PROGRAM Agitadores
VAR
	PP1_L1_AG: Equipo_Motor_No_Rev;
	wPP1_L1_AG_HoraIni:INT;
	wPP1_L1_AG_CantHora:INT;
	wPP1_L1_AG_HoraFin:INT;
	bPP1_L1_AG_ResetAl: BOOL;	
	//
	PP1_L2_AG: Equipo_Motor_No_Rev;
	wPP1_L2_AG_HoraIni:INT;
	wPP1_L2_AG_CantHora:INT;
	wPP1_L2_AG_HoraFin:INT;
	//
	PP1_L3_AG: Equipo_Motor_No_Rev;
	wPP1_L3_AG_HoraIni:INT;
	wPP1_L3_AG_CantHora:INT;
	wPP1_L3_AG_HoraFin:INT;	
	//
	PP1_L4_AG: Equipo_Motor_No_Rev;
	wPP1_L4_AG_HoraIni:INT;
	wPP1_L4_AG_CantHora:INT;
	wPP1_L4_AG_HoraFin:INT;	
	//	
	PP2_L5_AG: Equipo_Motor_No_Rev;
	wPP2_L5_AG_HoraIni:INT;
	wPP2_L5_AG_CantHora:INT;
	wPP2_L5_AG_HoraFin:INT;
	bPP2_L5_AG_ResetAl: BOOL;	
	//
	PP2_L6_AG: Equipo_Motor_No_Rev;
	wPP2_L6_AG_HoraIni:INT;
	wPP2_L6_AG_CantHora:INT;
	wPP2_L6_AG_HoraFin:INT;	
	//
	PP2_L7_AG: Equipo_Motor_No_Rev;
	wPP2_L7_AG_HoraIni:INT;
	wPP2_L7_AG_CantHora:INT;
	wPP2_L7_AG_HoraFin:INT;	
	//
	PP2_L8_AG: Equipo_Motor_No_Rev;
	wPP2_L8_AG_HoraIni:INT;
	wPP2_L8_AG_CantHora:INT;
	wPP2_L8_AG_HoraFin:INT;
	//
	PP3_L9_AG: Equipo_Motor_No_Rev;
	wPP3_L9_AG_HoraIni:INT;
	wPP3_L9_AG_CantHora:INT;
	wPP3_L9_AG_HoraFin:INT;	
	//
	PP3_L10_AG: Equipo_Motor_No_Rev;
	wPP3_L10_AG_HoraIni:INT;
	wPP3_L10_AG_CantHora:INT;
	wPP3_L10_AG_HoraFin:INT;	
	//
	PP3_L11_AG: Equipo_Motor_No_Rev;
	wPP3_L11_AG_HoraIni:INT;
	wPP3_L11_AG_CantHora:INT;
	wPP3_L11_AG_HoraFin:INT;	
	//
	PP3_L12_AG: Equipo_Motor_No_Rev;
	wPP3_L12_AG_HoraIni:INT;
	wPP3_L12_AG_CantHora:INT;
	wPP3_L12_AG_HoraFin:INT;	
END_VAR

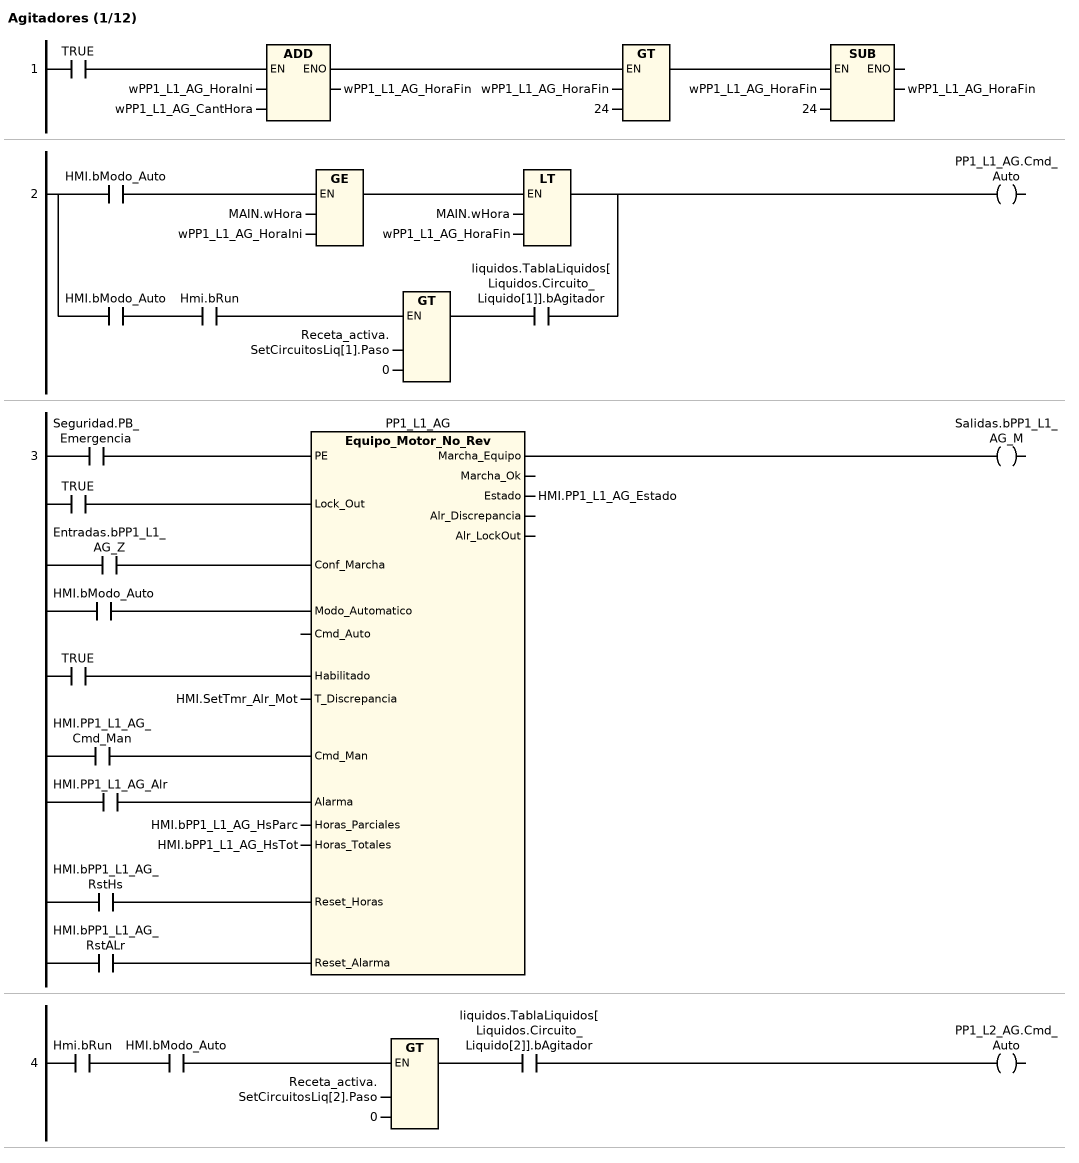
// NETWORK 1
wPP1_L1_AG_HoraFin := wPP1_L1_AG_HoraIni + wPP1_L1_AG_CantHora;
IF wPP1_L1_AG_HoraFin > 24 THEN wPP1_L1_AG_HoraFin := wPP1_L1_AG_HoraFin - 24; END_IF

// NETWORK 2
PP1_L1_AG.Cmd_Auto := HMI.bModo_Auto AND MAIN.wHora >= wPP1_L1_AG_HoraIni AND MAIN.wHora < wPP1_L1_AG_HoraFin OR (HMI.bModo_Auto AND Hmi.bRun AND Receta_activa.SetCircuitosLiq[1].Paso > 0) AND (liquidos.TablaLiquidos[Liquidos.Circuito_Liquido[1]].bAgitador);

// NETWORK 3
PP1_L1_AG(
    PE := Seguridad.PB_Emergencia,
    Lock_Out := TRUE,
    Conf_Marcha := Entradas.bPP1_L1_AG_Z,
    Modo_Automatico := HMI.bModo_Auto,
    Habilitado := TRUE,
    T_Discrepancia := HMI.SetTmr_Alr_Mot,
    Cmd_Man := HMI.PP1_L1_AG_Cmd_Man,
    Alarma := HMI.PP1_L1_AG_Alr,
    Horas_Parciales := HMI.bPP1_L1_AG_HsParc,
    Horas_Totales := HMI.bPP1_L1_AG_HsTot,
    Reset_Horas := HMI.bPP1_L1_AG_RstHs,
    Reset_Alarma := HMI.bPP1_L1_AG_RstALr,
    Estado => HMI.PP1_L1_AG_Estado); // Equipo_Motor_No_Rev
Salidas.bPP1_L1_AG_M := PP1_L1_AG.Marcha_Equipo;

// NETWORK 4
PP1_L2_AG.Cmd_Auto := (Hmi.bRun AND HMI.bModo_Auto AND Receta_activa.SetCircuitosLiq[2].Paso > 0) AND (liquidos.TablaLiquidos[Liquidos.Circuito_Liquido[2]].bAgitador);

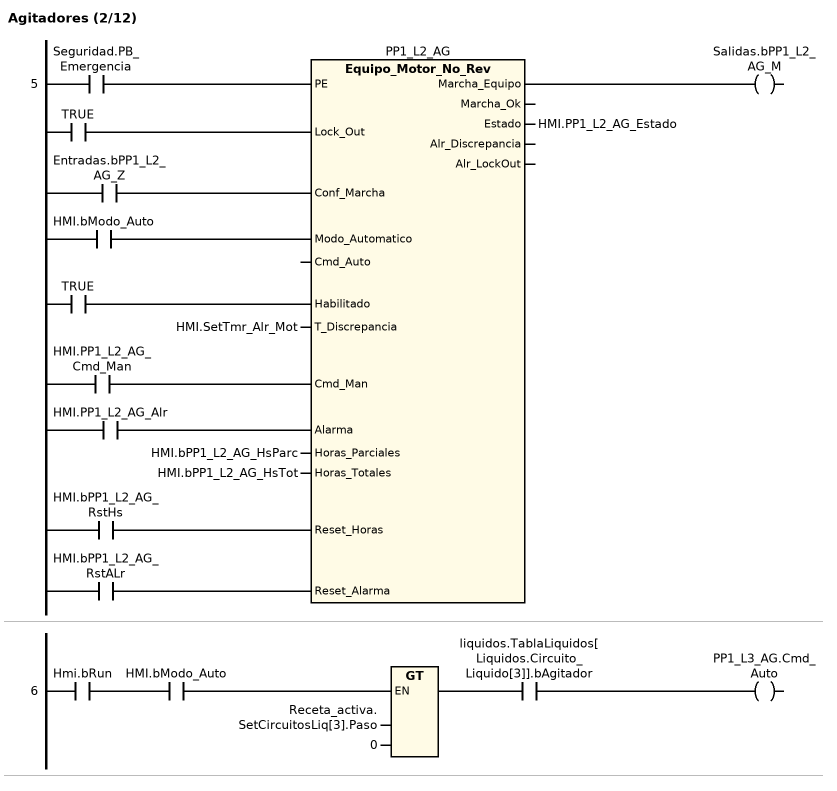
// NETWORK 5
PP1_L2_AG(
    PE := Seguridad.PB_Emergencia,
    Lock_Out := TRUE,
    Conf_Marcha := Entradas.bPP1_L2_AG_Z,
    Modo_Automatico := HMI.bModo_Auto,
    Habilitado := TRUE,
    T_Discrepancia := HMI.SetTmr_Alr_Mot,
    Cmd_Man := HMI.PP1_L2_AG_Cmd_Man,
    Alarma := HMI.PP1_L2_AG_Alr,
    Horas_Parciales := HMI.bPP1_L2_AG_HsParc,
    Horas_Totales := HMI.bPP1_L2_AG_HsTot,
    Reset_Horas := HMI.bPP1_L2_AG_RstHs,
    Reset_Alarma := HMI.bPP1_L2_AG_RstALr,
    Estado => HMI.PP1_L2_AG_Estado); // Equipo_Motor_No_Rev
Salidas.bPP1_L2_AG_M := PP1_L2_AG.Marcha_Equipo;

// NETWORK 6
PP1_L3_AG.Cmd_Auto := (Hmi.bRun AND HMI.bModo_Auto AND Receta_activa.SetCircuitosLiq[3].Paso > 0) AND (liquidos.TablaLiquidos[Liquidos.Circuito_Liquido[3]].bAgitador);

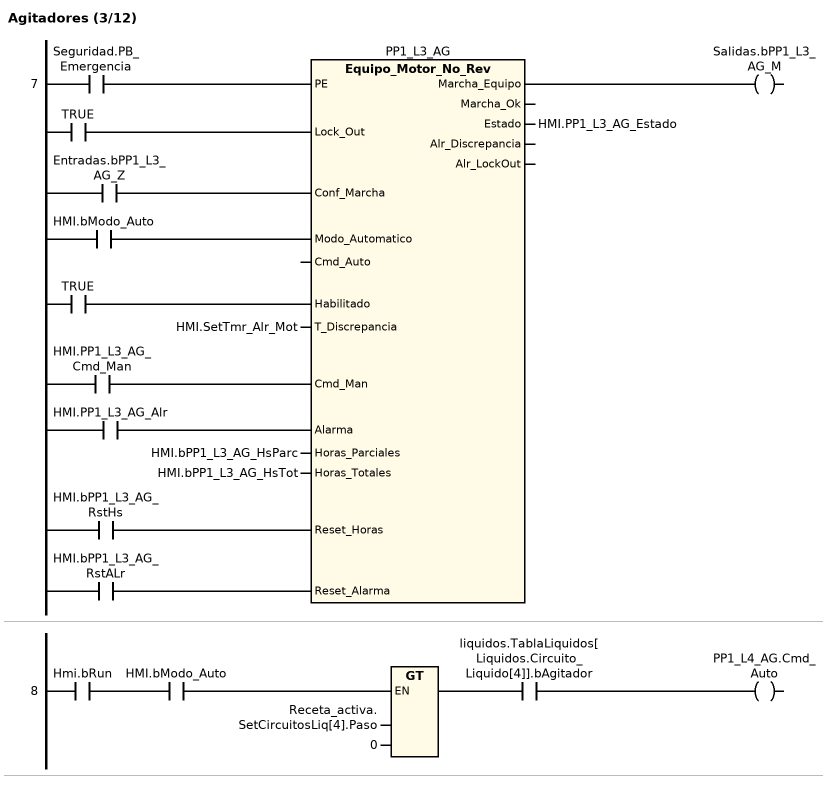
// NETWORK 7
PP1_L3_AG(
    PE := Seguridad.PB_Emergencia,
    Lock_Out := TRUE,
    Conf_Marcha := Entradas.bPP1_L3_AG_Z,
    Modo_Automatico := HMI.bModo_Auto,
    Habilitado := TRUE,
    T_Discrepancia := HMI.SetTmr_Alr_Mot,
    Cmd_Man := HMI.PP1_L3_AG_Cmd_Man,
    Alarma := HMI.PP1_L3_AG_Alr,
    Horas_Parciales := HMI.bPP1_L3_AG_HsParc,
    Horas_Totales := HMI.bPP1_L3_AG_HsTot,
    Reset_Horas := HMI.bPP1_L3_AG_RstHs,
    Reset_Alarma := HMI.bPP1_L3_AG_RstALr,
    Estado => HMI.PP1_L3_AG_Estado); // Equipo_Motor_No_Rev
Salidas.bPP1_L3_AG_M := PP1_L3_AG.Marcha_Equipo;

// NETWORK 8
PP1_L4_AG.Cmd_Auto := (Hmi.bRun AND HMI.bModo_Auto AND Receta_activa.SetCircuitosLiq[4].Paso > 0) AND (liquidos.TablaLiquidos[Liquidos.Circuito_Liquido[4]].bAgitador);

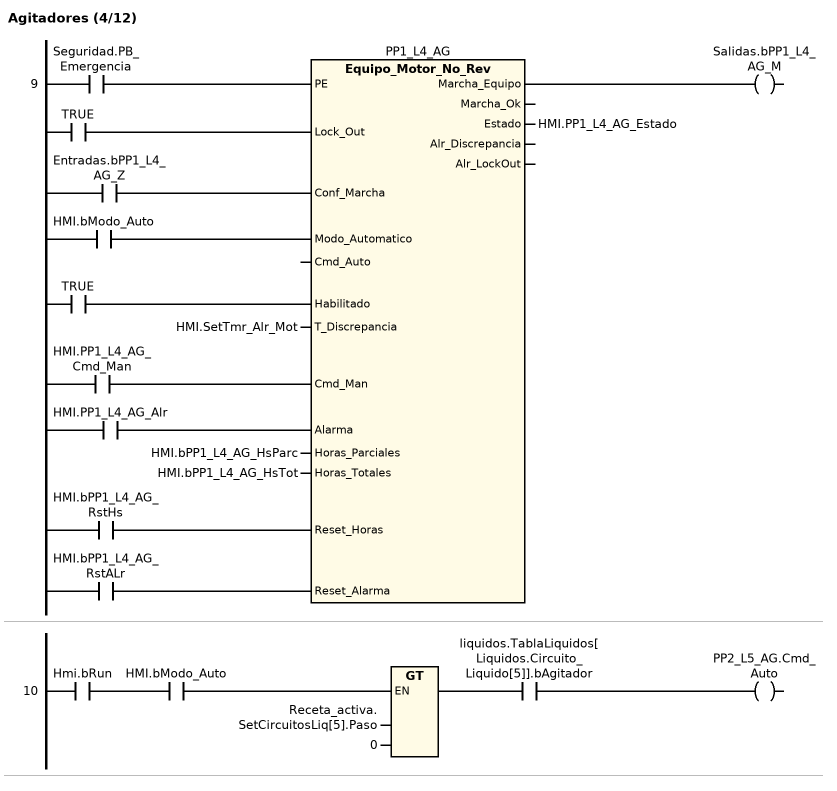
// NETWORK 9
PP1_L4_AG(
    PE := Seguridad.PB_Emergencia,
    Lock_Out := TRUE,
    Conf_Marcha := Entradas.bPP1_L4_AG_Z,
    Modo_Automatico := HMI.bModo_Auto,
    Habilitado := TRUE,
    T_Discrepancia := HMI.SetTmr_Alr_Mot,
    Cmd_Man := HMI.PP1_L4_AG_Cmd_Man,
    Alarma := HMI.PP1_L4_AG_Alr,
    Horas_Parciales := HMI.bPP1_L4_AG_HsParc,
    Horas_Totales := HMI.bPP1_L4_AG_HsTot,
    Reset_Horas := HMI.bPP1_L4_AG_RstHs,
    Reset_Alarma := HMI.bPP1_L4_AG_RstALr,
    Estado => HMI.PP1_L4_AG_Estado); // Equipo_Motor_No_Rev
Salidas.bPP1_L4_AG_M := PP1_L4_AG.Marcha_Equipo;

// NETWORK 10
PP2_L5_AG.Cmd_Auto := (Hmi.bRun AND HMI.bModo_Auto AND Receta_activa.SetCircuitosLiq[5].Paso > 0) AND (liquidos.TablaLiquidos[Liquidos.Circuito_Liquido[5]].bAgitador);

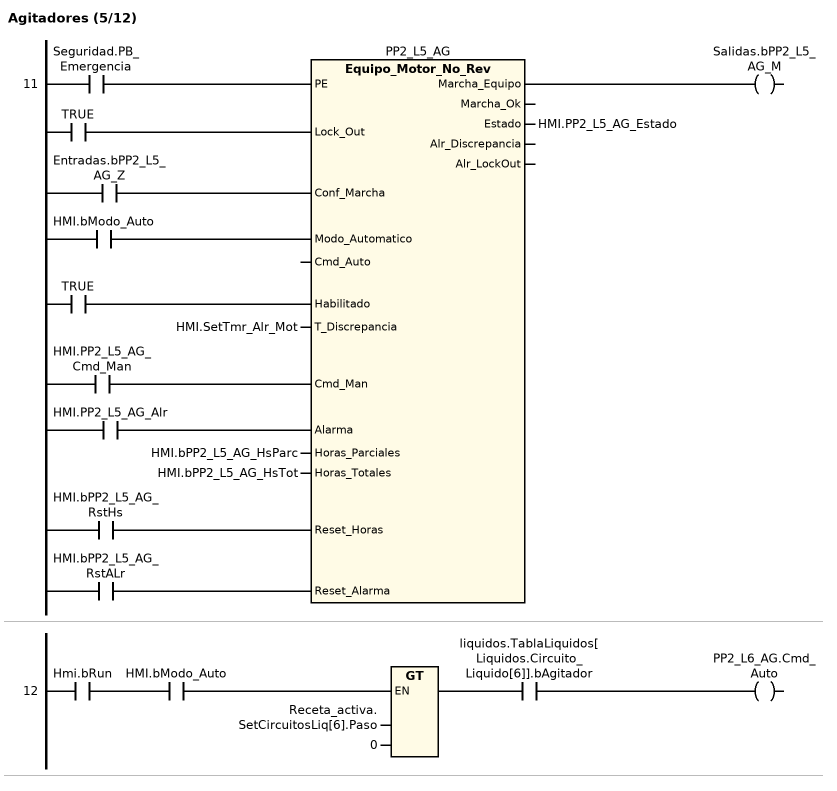
// NETWORK 11
PP2_L5_AG(
    PE := Seguridad.PB_Emergencia,
    Lock_Out := TRUE,
    Conf_Marcha := Entradas.bPP2_L5_AG_Z,
    Modo_Automatico := HMI.bModo_Auto,
    Habilitado := TRUE,
    T_Discrepancia := HMI.SetTmr_Alr_Mot,
    Cmd_Man := HMI.PP2_L5_AG_Cmd_Man,
    Alarma := HMI.PP2_L5_AG_Alr,
    Horas_Parciales := HMI.bPP2_L5_AG_HsParc,
    Horas_Totales := HMI.bPP2_L5_AG_HsTot,
    Reset_Horas := HMI.bPP2_L5_AG_RstHs,
    Reset_Alarma := HMI.bPP2_L5_AG_RstALr,
    Estado => HMI.PP2_L5_AG_Estado); // Equipo_Motor_No_Rev
Salidas.bPP2_L5_AG_M := PP2_L5_AG.Marcha_Equipo;

// NETWORK 12
PP2_L6_AG.Cmd_Auto := (Hmi.bRun AND HMI.bModo_Auto AND Receta_activa.SetCircuitosLiq[6].Paso > 0) AND (liquidos.TablaLiquidos[Liquidos.Circuito_Liquido[6]].bAgitador);

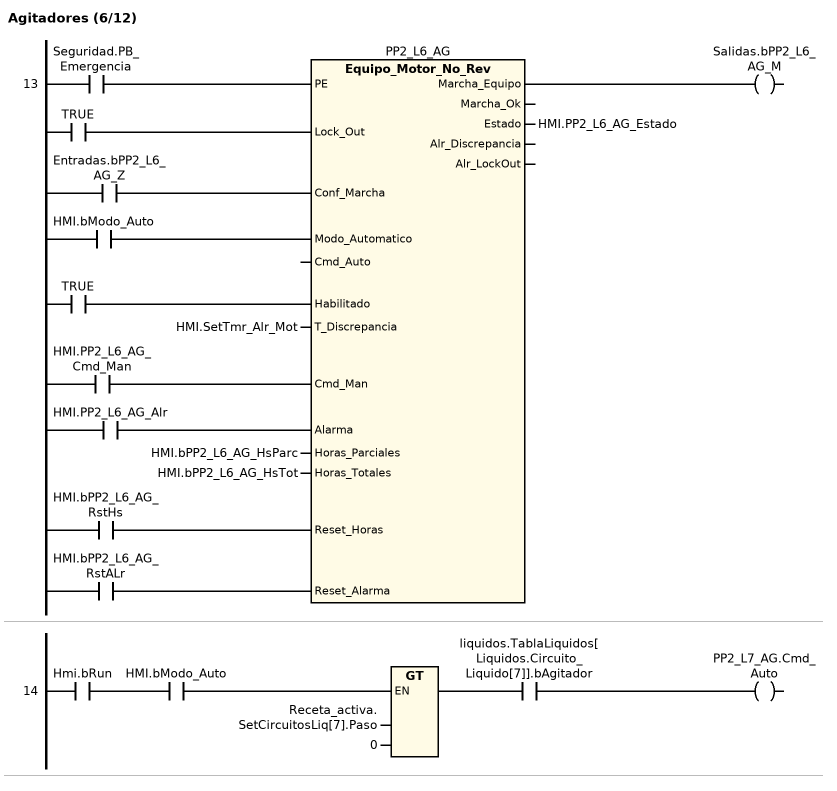
// NETWORK 13
PP2_L6_AG(
    PE := Seguridad.PB_Emergencia,
    Lock_Out := TRUE,
    Conf_Marcha := Entradas.bPP2_L6_AG_Z,
    Modo_Automatico := HMI.bModo_Auto,
    Habilitado := TRUE,
    T_Discrepancia := HMI.SetTmr_Alr_Mot,
    Cmd_Man := HMI.PP2_L6_AG_Cmd_Man,
    Alarma := HMI.PP2_L6_AG_Alr,
    Horas_Parciales := HMI.bPP2_L6_AG_HsParc,
    Horas_Totales := HMI.bPP2_L6_AG_HsTot,
    Reset_Horas := HMI.bPP2_L6_AG_RstHs,
    Reset_Alarma := HMI.bPP2_L6_AG_RstALr,
    Estado => HMI.PP2_L6_AG_Estado); // Equipo_Motor_No_Rev
Salidas.bPP2_L6_AG_M := PP2_L6_AG.Marcha_Equipo;

// NETWORK 14
PP2_L7_AG.Cmd_Auto := (Hmi.bRun AND HMI.bModo_Auto AND Receta_activa.SetCircuitosLiq[7].Paso > 0) AND (liquidos.TablaLiquidos[Liquidos.Circuito_Liquido[7]].bAgitador);

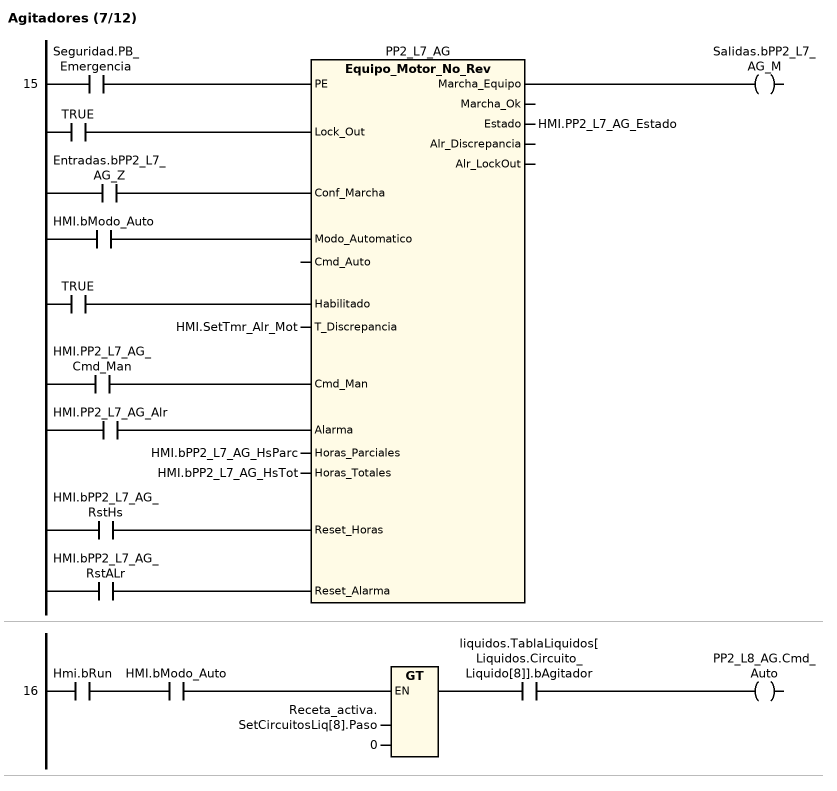
// NETWORK 15
PP2_L7_AG(
    PE := Seguridad.PB_Emergencia,
    Lock_Out := TRUE,
    Conf_Marcha := Entradas.bPP2_L7_AG_Z,
    Modo_Automatico := HMI.bModo_Auto,
    Habilitado := TRUE,
    T_Discrepancia := HMI.SetTmr_Alr_Mot,
    Cmd_Man := HMI.PP2_L7_AG_Cmd_Man,
    Alarma := HMI.PP2_L7_AG_Alr,
    Horas_Parciales := HMI.bPP2_L7_AG_HsParc,
    Horas_Totales := HMI.bPP2_L7_AG_HsTot,
    Reset_Horas := HMI.bPP2_L7_AG_RstHs,
    Reset_Alarma := HMI.bPP2_L7_AG_RstALr,
    Estado => HMI.PP2_L7_AG_Estado); // Equipo_Motor_No_Rev
Salidas.bPP2_L7_AG_M := PP2_L7_AG.Marcha_Equipo;

// NETWORK 16
PP2_L8_AG.Cmd_Auto := (Hmi.bRun AND HMI.bModo_Auto AND Receta_activa.SetCircuitosLiq[8].Paso > 0) AND (liquidos.TablaLiquidos[Liquidos.Circuito_Liquido[8]].bAgitador);

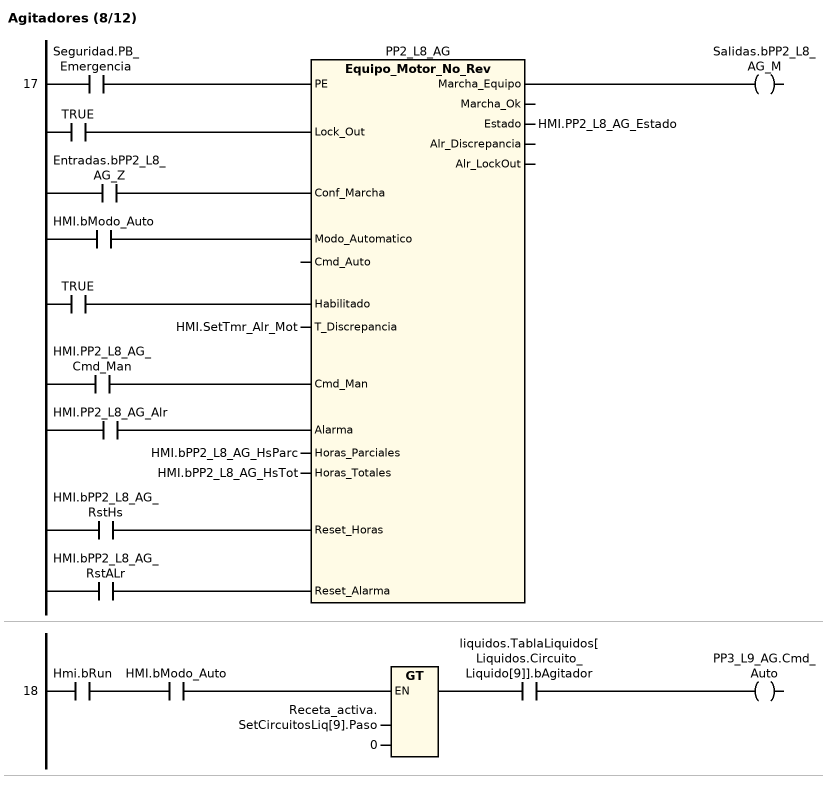
// NETWORK 17
PP2_L8_AG(
    PE := Seguridad.PB_Emergencia,
    Lock_Out := TRUE,
    Conf_Marcha := Entradas.bPP2_L8_AG_Z,
    Modo_Automatico := HMI.bModo_Auto,
    Habilitado := TRUE,
    T_Discrepancia := HMI.SetTmr_Alr_Mot,
    Cmd_Man := HMI.PP2_L8_AG_Cmd_Man,
    Alarma := HMI.PP2_L8_AG_Alr,
    Horas_Parciales := HMI.bPP2_L8_AG_HsParc,
    Horas_Totales := HMI.bPP2_L8_AG_HsTot,
    Reset_Horas := HMI.bPP2_L8_AG_RstHs,
    Reset_Alarma := HMI.bPP2_L8_AG_RstALr,
    Estado => HMI.PP2_L8_AG_Estado); // Equipo_Motor_No_Rev
Salidas.bPP2_L8_AG_M := PP2_L8_AG.Marcha_Equipo;

// NETWORK 18
PP3_L9_AG.Cmd_Auto := (Hmi.bRun AND HMI.bModo_Auto AND Receta_activa.SetCircuitosLiq[9].Paso > 0) AND (liquidos.TablaLiquidos[Liquidos.Circuito_Liquido[9]].bAgitador);

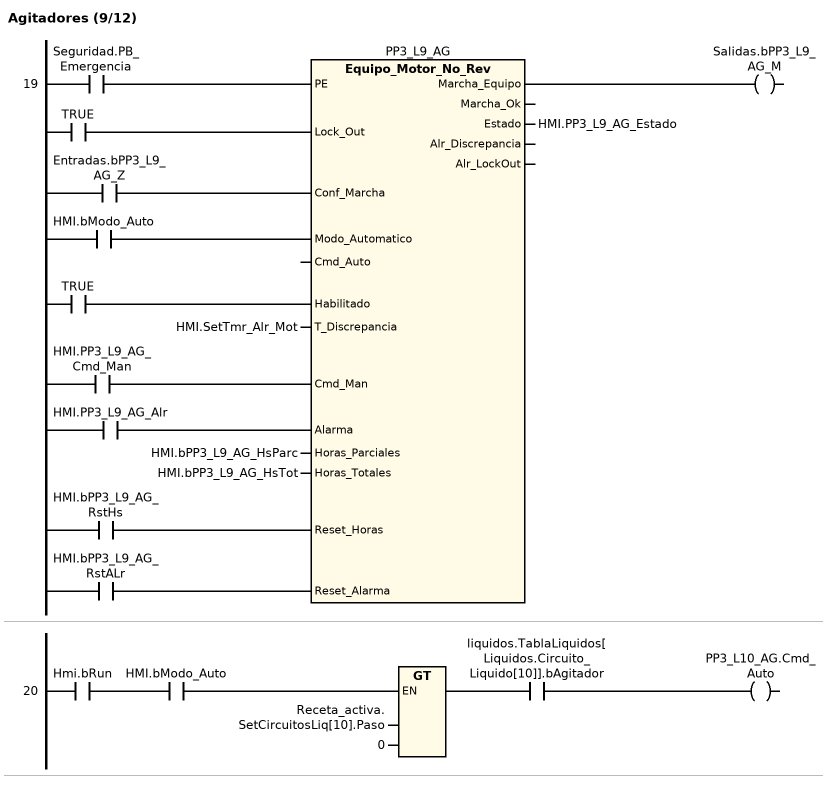
// NETWORK 19
PP3_L9_AG(
    PE := Seguridad.PB_Emergencia,
    Lock_Out := TRUE,
    Conf_Marcha := Entradas.bPP3_L9_AG_Z,
    Modo_Automatico := HMI.bModo_Auto,
    Habilitado := TRUE,
    T_Discrepancia := HMI.SetTmr_Alr_Mot,
    Cmd_Man := HMI.PP3_L9_AG_Cmd_Man,
    Alarma := HMI.PP3_L9_AG_Alr,
    Horas_Parciales := HMI.bPP3_L9_AG_HsParc,
    Horas_Totales := HMI.bPP3_L9_AG_HsTot,
    Reset_Horas := HMI.bPP3_L9_AG_RstHs,
    Reset_Alarma := HMI.bPP3_L9_AG_RstALr,
    Estado => HMI.PP3_L9_AG_Estado); // Equipo_Motor_No_Rev
Salidas.bPP3_L9_AG_M := PP3_L9_AG.Marcha_Equipo;

// NETWORK 20
PP3_L10_AG.Cmd_Auto := (Hmi.bRun AND HMI.bModo_Auto AND Receta_activa.SetCircuitosLiq[10].Paso > 0) AND (liquidos.TablaLiquidos[Liquidos.Circuito_Liquido[10]].bAgitador);

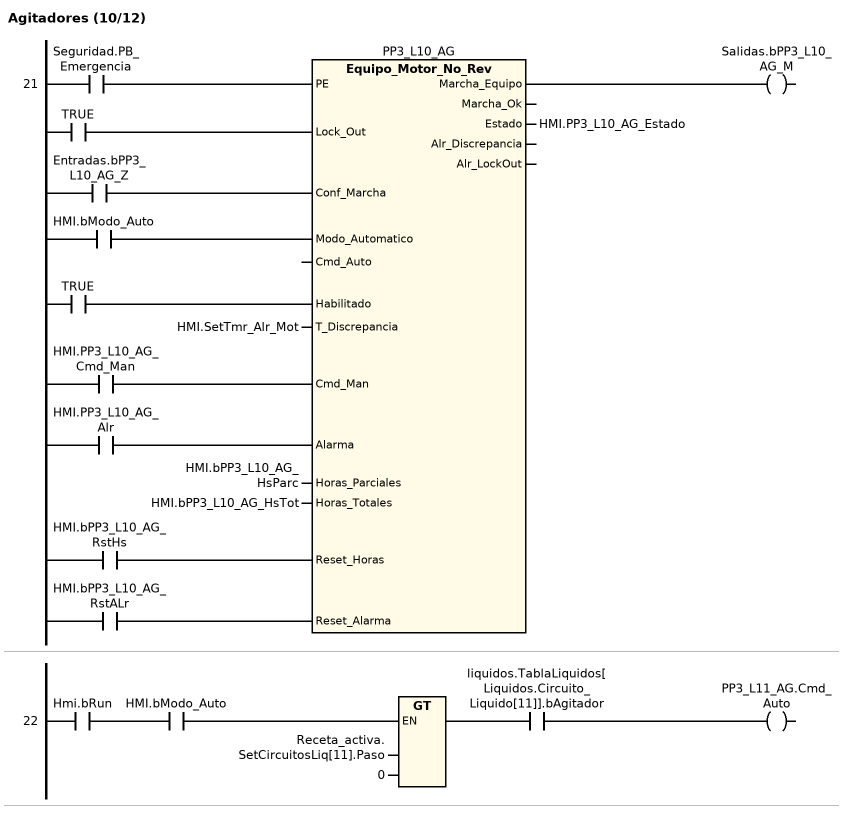
// NETWORK 21
PP3_L10_AG(
    PE := Seguridad.PB_Emergencia,
    Lock_Out := TRUE,
    Conf_Marcha := Entradas.bPP3_L10_AG_Z,
    Modo_Automatico := HMI.bModo_Auto,
    Habilitado := TRUE,
    T_Discrepancia := HMI.SetTmr_Alr_Mot,
    Cmd_Man := HMI.PP3_L10_AG_Cmd_Man,
    Alarma := HMI.PP3_L10_AG_Alr,
    Horas_Parciales := HMI.bPP3_L10_AG_HsParc,
    Horas_Totales := HMI.bPP3_L10_AG_HsTot,
    Reset_Horas := HMI.bPP3_L10_AG_RstHs,
    Reset_Alarma := HMI.bPP3_L10_AG_RstALr,
    Estado => HMI.PP3_L10_AG_Estado); // Equipo_Motor_No_Rev
Salidas.bPP3_L10_AG_M := PP3_L10_AG.Marcha_Equipo;

// NETWORK 22
PP3_L11_AG.Cmd_Auto := (Hmi.bRun AND HMI.bModo_Auto AND Receta_activa.SetCircuitosLiq[11].Paso > 0) AND (liquidos.TablaLiquidos[Liquidos.Circuito_Liquido[11]].bAgitador);

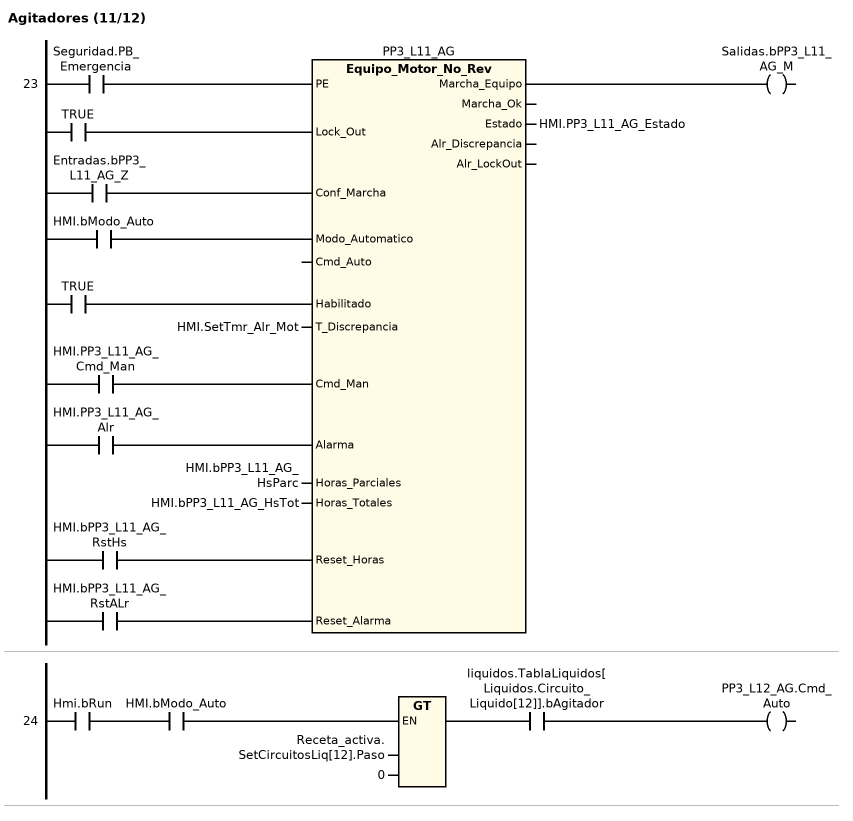
// NETWORK 23
PP3_L11_AG(
    PE := Seguridad.PB_Emergencia,
    Lock_Out := TRUE,
    Conf_Marcha := Entradas.bPP3_L11_AG_Z,
    Modo_Automatico := HMI.bModo_Auto,
    Habilitado := TRUE,
    T_Discrepancia := HMI.SetTmr_Alr_Mot,
    Cmd_Man := HMI.PP3_L11_AG_Cmd_Man,
    Alarma := HMI.PP3_L11_AG_Alr,
    Horas_Parciales := HMI.bPP3_L11_AG_HsParc,
    Horas_Totales := HMI.bPP3_L11_AG_HsTot,
    Reset_Horas := HMI.bPP3_L11_AG_RstHs,
    Reset_Alarma := HMI.bPP3_L11_AG_RstALr,
    Estado => HMI.PP3_L11_AG_Estado); // Equipo_Motor_No_Rev
Salidas.bPP3_L11_AG_M := PP3_L11_AG.Marcha_Equipo;

// NETWORK 24
PP3_L12_AG.Cmd_Auto := (Hmi.bRun AND HMI.bModo_Auto AND Receta_activa.SetCircuitosLiq[12].Paso > 0) AND (liquidos.TablaLiquidos[Liquidos.Circuito_Liquido[12]].bAgitador);

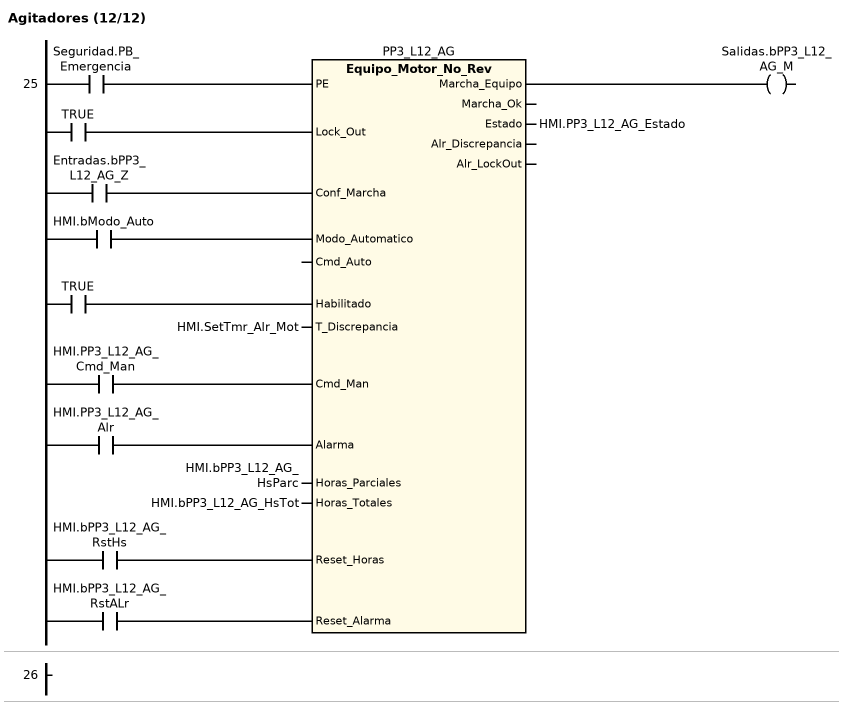
// NETWORK 25
PP3_L12_AG(
    PE := Seguridad.PB_Emergencia,
    Lock_Out := TRUE,
    Conf_Marcha := Entradas.bPP3_L12_AG_Z,
    Modo_Automatico := HMI.bModo_Auto,
    Habilitado := TRUE,
    T_Discrepancia := HMI.SetTmr_Alr_Mot,
    Cmd_Man := HMI.PP3_L12_AG_Cmd_Man,
    Alarma := HMI.PP3_L12_AG_Alr,
    Horas_Parciales := HMI.bPP3_L12_AG_HsParc,
    Horas_Totales := HMI.bPP3_L12_AG_HsTot,
    Reset_Horas := HMI.bPP3_L12_AG_RstHs,
    Reset_Alarma := HMI.bPP3_L12_AG_RstALr,
    Estado => HMI.PP3_L12_AG_Estado); // Equipo_Motor_No_Rev
Salidas.bPP3_L12_AG_M := PP3_L12_AG.Marcha_Equipo;

// NETWORK 26

END_PROGRAM

(* stored: Version 1.1.0.1, ProductVersion 3.1.4024.14
   POU Agitadores: Id {c1657423-0305-49c7-aaf6-a3ab77aeb1b0}, SpecialFunc None *)
